TYPE MoveState_t :
(
	MOVESTATE_INIT,
	MOVESTATE_ENABLE,
	MOVESTATE_FORWARD,
	MOVESTATE_CAMIN,
	MOVESTATE_SWITCHCAM,
	MOVESTATE_READCAMDATA,
	MOVESTATE_PREPARECAMMODIFICATION,
	MOVESTATE_MODIFYCAM,
	MOVESTATE_CAMSCALING,
	MOVESTATE_CAMOUT,
	MOVESTATE_STOPMASTER,
	MOVESTATE_STOPAXES,
	MOVESTATE_ERROR,
	MOVESTATE_RESET
) UDINT;
END_TYPE

(* stored: Version 1.1.0.1, ProductVersion 3.1.4018.5
   DUT MoveState_t: Id {a8802f66-1f97-4eae-9c7d-b537add07402} *)
